# EPICS substitutions: odmApp/Db/bkh_odm_supervisor.substitutions
file bkhBi_simple.db {
pattern
    {ADDR,          ATTR,     DESC,         PORT,      ZSV,      OSV}
    {   0, :1104_01_CH01, "Chan01", $(M)_1104_01, NO_ALARM, NO_ALARM}
    {   1, :1104_01_CH02, "Chan02", $(M)_1104_01, NO_ALARM, NO_ALARM}
    {   2, :1104_01_CH03, "Chan03", $(M)_1104_01, NO_ALARM, NO_ALARM}
    {   3, :1104_01_CH04, "Chan04", $(M)_1104_01, NO_ALARM, NO_ALARM}
    {   4, :1104_01_CH05, "Chan05", $(M)_1104_01, NO_ALARM, NO_ALARM}
    {   5, :1104_01_CH06, "Chan06", $(M)_1104_01, NO_ALARM, NO_ALARM}
    {   6, :1104_01_CH07, "Chan07", $(M)_1104_01, NO_ALARM, NO_ALARM}
    {   7, :1104_01_CH08, "Chan08", $(M)_1104_01, NO_ALARM, NO_ALARM}
    {   8, :1104_01_CH09, "Chan09", $(M)_1104_01, NO_ALARM, NO_ALARM}
    {   9, :1104_01_CH10, "Chan10", $(M)_1104_01, NO_ALARM, NO_ALARM}
    {  10, :1104_01_CH11, "Chan11", $(M)_1104_01, NO_ALARM, NO_ALARM}
    {  11, :1104_01_CH12, "Chan12", $(M)_1104_01, NO_ALARM, NO_ALARM}
    {  12, :1104_01_CH13, "Chan13", $(M)_1104_01, NO_ALARM, NO_ALARM}
    {  13, :1104_01_CH14, "Chan14", $(M)_1104_01, NO_ALARM, NO_ALARM}
    {  14, :1104_01_CH15, "Chan15", $(M)_1104_01, NO_ALARM, NO_ALARM}
    {  15, :1104_01_CH16, "Chan16", $(M)_1104_01, NO_ALARM, NO_ALARM}
    {  16, :1104_01_CH17, "Chan17", $(M)_1104_01, NO_ALARM, NO_ALARM}
    {  17, :1104_01_CH18, "Chan18", $(M)_1104_01, NO_ALARM, NO_ALARM}
    {  18, :1104_01_CH19, "Chan19", $(M)_1104_01, NO_ALARM, NO_ALARM}
    {  19, :1104_01_CH20, "Chan20", $(M)_1104_01, NO_ALARM, NO_ALARM}
    {  20, :1104_01_CH21, "Chan21", $(M)_1104_01, NO_ALARM, NO_ALARM}
    {  21, :1104_01_CH22, "Chan22", $(M)_1104_01, NO_ALARM, NO_ALARM}
    {  22, :1104_01_CH23, "Chan23", $(M)_1104_01, NO_ALARM, NO_ALARM}
    {  23, :1104_01_CH24, "Chan24", $(M)_1104_01, NO_ALARM, NO_ALARM}
    {  24, :1104_01_CH25, "Chan25", $(M)_1104_01, NO_ALARM, NO_ALARM}
    {  25, :1104_01_CH26, "Chan26", $(M)_1104_01, NO_ALARM, NO_ALARM}
    {  26, :1104_01_CH27, "Chan27", $(M)_1104_01, NO_ALARM, NO_ALARM}
    {  27, :1104_01_CH28, "Chan28", $(M)_1104_01, NO_ALARM, NO_ALARM}
    {  28, :1104_01_CH29, "Chan29", $(M)_1104_01, NO_ALARM, NO_ALARM}
    {  29, :1104_01_CH30, "Chan30", $(M)_1104_01, NO_ALARM, NO_ALARM}
    {  30, :1104_01_CH31, "Chan31", $(M)_1104_01, NO_ALARM, NO_ALARM}
    {  31, :1104_01_CH32, "Chan32", $(M)_1104_01, NO_ALARM, NO_ALARM}
    {  32, :1104_01_CH33, "Chan33", $(M)_1104_01, NO_ALARM, NO_ALARM}
    {  33, :1104_01_CH34, "Chan34", $(M)_1104_01, NO_ALARM, NO_ALARM}
}

file bkhBo_simple.db {
pattern
    {ADDR,          ATTR,     DESC,         PORT}
    {   0, :2114_01_CH01, "Chan01", $(M)_2114_01}
    {   1, :2114_01_CH02, "Chan02", $(M)_2114_01}
    {   2, :2114_01_CH03, "Chan03", $(M)_2114_01}
    {   3, :2114_01_CH04, "Chan04", $(M)_2114_01}
}

# Not needed for digitial I/O modules
#file readwrite.db {
#pattern
#    {    MOD,         PORT}
#    {3012_01, $(M)_3012_01}
#}

file bkhAErr.db {
pattern
    {    MOD,         PORT}
    {1104_01, $(M)_1104_01}
    {2114_01, $(M)_2114_01}
}

# For bus coupler
file bk9000.db {
pattern
    {     DPORT,        RPORT,        WPORT}
    {$(M)_DEBUG, $(M)_BK9000R, $(M)_BK9000W}
}

file asynRecord.db {
pattern
    {      R, PORT, ADDR, IMAX, OMAX}
    {":Asyn", $(M),    0,    0,    0}
}

file statistics.template {
pattern
    {        R, PORT,        SCAN}
    {":Modbus", $(M), "10 second"}
}
